{attribute 'Tc2GvlVarNames'}
{attribute 'strict'}
//Stato Operazione LGV
TYPE e_Stato_Operazione_LGV :
(
	LGV_OPERAZIONE_VERIFICATA 	:= 0,	(* Indica che l'operazione svolta da parte del veicolo è stata verificata *)
	LGV_PRELIEVO_EFFETTUATO 	:= 1,	(* Indica che il prelievo da parte del veicolo è stato effettuato *)   
	LGV_DEPOSITO_EFFETTUATO 	:= 2	(* Indica che il deposito da parte del veicolo è stato effettuato *)
);
END_TYPE

(* stored: Version 1.1.0.1, ProductVersion 3.1.4022.10
   EnumerationTextList e_Stato_Operazione_LGV: Id {f5d74f5b-792e-40d3-804f-3aa70597ee7e} *)
